(* Logix 5000 project; controller WASH_TON Emulate 5570 rev 36.11; software revision 36.00 *)

TASK MainTask (continuous, watchdog 500 ms) : MainProgram, Model

MODULES
   Local : Emulate 5570 (ICP 2, rev 36.11)
       : 1756-IB16 (ICP 3, rev 3.1, Input RPI 20 ms)
       : vendor 1 type 7 code 16 (ICP 4, rev 3.1, Output RPI 20 ms)
END_MODULES

VAR_GLOBAL   (* controller tags *)
   PUSHBUTTON : ALIAS FOR Local:3:I.Data.0;   // Pushbutton Wash Cycle
   SOLENOID_CLAMP1 : ALIAS FOR Local:4:O.Data.0;   // Clamp 1 Solenoid
   SOLENOID_CLAMP2 : ALIAS FOR Local:4:O.Data.1;   // Clamp 2 Solenoid
   SWITCH_CLAMP1 : ALIAS FOR Local:3:I.Data.1;   // Limit Switch Clamp 1
   SWITCH_CLAMP2 : ALIAS FOR Local:3:I.Data.2;   // Limit Switch Clamp 2
   WASH_VALVE : ALIAS FOR Local:4:O.Data.2;   // Spray Wash Valve
END_VAR

PROGRAM MainProgram   (* main routine FuncRoutine *)
VAR
   BAND_01 : FBD_BOOLEAN_AND := (In4 := 1, In5 := 1, In6 := 1, In7 := 1, In8 := 1);
   BAND_02 : FBD_BOOLEAN_AND := (In4 := 1, In5 := 1, In6 := 1, In7 := 1, In8 := 1);
   BNOT_01 : FBD_BOOLEAN_NOT := (Out := 1);
   WASH_TIMER : FBD_TIMER := (PRE := 3000);
END_VAR

ROUTINE FuncRoutine   (* function block diagram *)
   SHEET 1
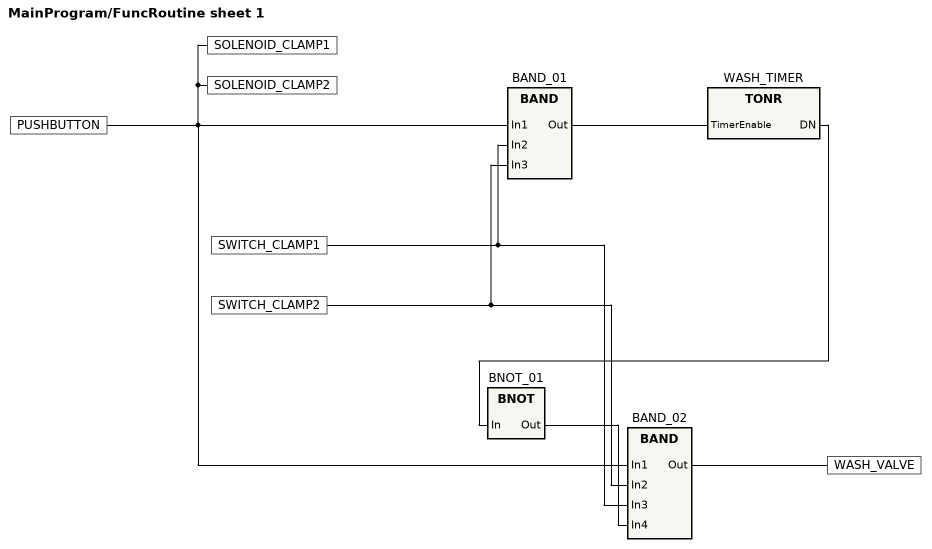
   SOLENOID_CLAMP1 := PUSHBUTTON;
   SOLENOID_CLAMP2 := PUSHBUTTON;
   BAND_01 : BAND(In1 := PUSHBUTTON, In2 := SWITCH_CLAMP1, In3 := SWITCH_CLAMP2);
   WASH_TIMER : TONR(TimerEnable := BAND_01.Out);
   BNOT_01 : BNOT(In := WASH_TIMER.DN);
   BAND_02 : BAND(In1 := PUSHBUTTON, In2 := SWITCH_CLAMP2, In3 := SWITCH_CLAMP1, In4 := BNOT_01.Out);
   WASH_VALVE := BAND_02.Out;
END_ROUTINE
END_PROGRAM

PROGRAM Model   (* main routine Emulate *)
VAR
   HOLD : DINT;
   SOL_1_CLSD : TIMER := (PRE := 3000);
   SOL_1_OPN : TIMER := (PRE := 1000, ACC := 1000, EN := 1, DN := 1);
   SOL_2_CLSD : TIMER := (PRE := 1000);
   SOL_2_OPN : TIMER := (PRE := 2000, ACC := 2000, EN := 1, DN := 1);
END_VAR

ROUTINE Emulate   (* ladder *)
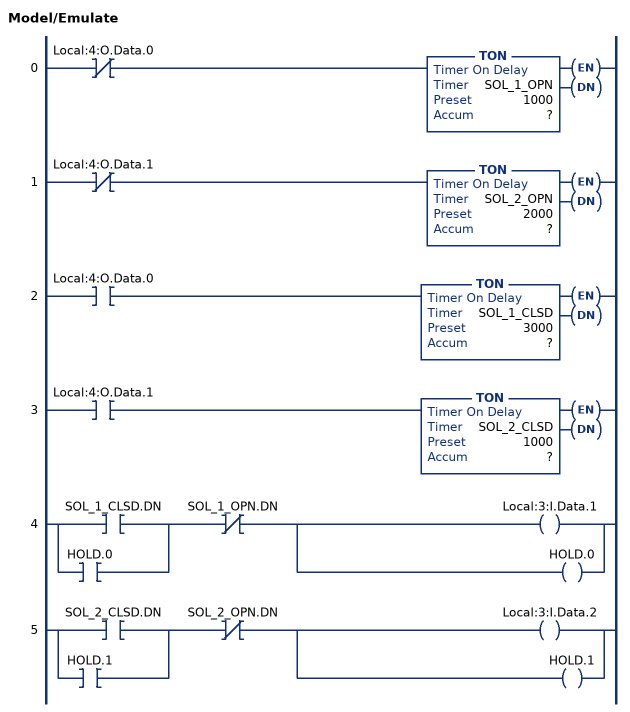
   0: XIO(Local:4:O.Data.0)TON(SOL_1_OPN,?,?);
   1: XIO(Local:4:O.Data.1)TON(SOL_2_OPN,?,?);
   2: XIC(Local:4:O.Data.0)TON(SOL_1_CLSD,?,?);
   3: XIC(Local:4:O.Data.1)TON(SOL_2_CLSD,?,?);
   4: [XIC(SOL_1_CLSD.DN) ,XIC(HOLD.0) ]XIO(SOL_1_OPN.DN)[OTE(Local:3:I.Data.1) ,OTE(HOLD.0) ];
   5: [XIC(SOL_2_CLSD.DN) ,XIC(HOLD.1) ]XIO(SOL_2_OPN.DN)[OTE(Local:3:I.Data.2) ,OTE(HOLD.1) ];
END_ROUTINE
END_PROGRAM
